// TIA Portal V18 export
TYPE "LGasp_TypeData_fromERP"
// stored: IsFailsafeCompliant false
   STRUCT
      operator : WString[30];   // Operatore loggato al sistema ERP del cliente
      coilsetup : Array[1..4] of "LGasp_TypeCoil_fromERP";
   END_STRUCT;
END_TYPE
